(* Logix 5000 project; controller Reto1 vendor 1 type 14 code 156 rev 30.11; software revision 30.00 *)

TASK MainTask (continuous, watchdog 500 ms) : MainProgram

MODULES
   Local : vendor 1 type 14 code 156 (Compact 0, rev 30.11)
END_MODULES

VAR_GLOBAL   (* controller tags *)
   C0 : BOOL;   // OK_INITIALIZATION
   C1 : BOOL;   // OK_STSTEM_ON
   C2 : BOOL;   // OK_POS_TAPA
   C3 : BOOL;   // OK_POS_BASE
   C4 : BOOL;   // OK_FORMADO
   C5 : BOOL;   // OK_FORMADO2
   C6 : BOOL;   // OK_RESET_PROCESS
   CONT_CAJAS : COUNTER := (PRE := 10);
   E0 : BOOL;   // INITIALIZATION
   E1 : BOOL;   // STSTEM_ON
   E2 : BOOL;   // POS_TAPA
   E3 : BOOL;   // POS_BASE
   E4 : BOOL;   // FORMADO
   E5 : BOOL;   // FORMADO2
   E6 : BOOL;   // RESET_PROCESS
   ENT_BASE : BOOL;
   ENT_LID : BOOL;
   ES : BOOL;   // Help Emergency Stop
   GD_IN_0 : BOOL;   // GD_MOVING_X
   GD_IN_1 : BOOL;   // GD_MOVING_Z
   GD_IN_10 : BOOL;   // START_ALL
   GD_IN_11 : BOOL;   // RESET
   GD_IN_12 : BOOL;   // STOP_ALL
   GD_IN_13 : BOOL;   // GD Emergency Stop
   GD_IN_2 : BOOL;   // ITEM_DETECTER
   GD_IN_3 : BOOL;   // LID_AT_PLACE
   GD_IN_4 : BOOL;   // GD_LID_CLAMPED
   GD_IN_5 : BOOL;   // POS_LIMIT_LIDS
   GD_IN_6 : BOOL;   // BASE_AT_PLACE
   GD_IN_7 : BOOL;   // GD_BASE_CLAMPED
   GD_IN_8 : BOOL;   // POS_LIMIT_BASES
   GD_IN_9 : BOOL;   // GD_PART_LEAVING
   GD_OUT_0 : BOOL;   // MOVE_X
   GD_OUT_1 : BOOL;   // MOVE_Z
   GD_OUT_10 : BOOL;   // RESET_LIGHT
   GD_OUT_11 : BOOL;   // STOP_LIGHT
   GD_OUT_2 : BOOL;   // GRAB
   GD_OUT_3 : BOOL;   // LIDS_CONVEYOR
   GD_OUT_4 : BOOL;   // CLAMP_LID
   GD_OUT_5 : BOOL;   // GD_LID_POS_RAISED
   GD_OUT_6 : BOOL;   // BASES_CONVEYOR
   GD_OUT_7 : BOOL;   // CLAMP_BASE
   GD_OUT_8 : BOOL;   // GD_BASE_POS_RAISED
   GD_OUT_9 : BOOL;   // START_LIGHT
   INT1 : BOOL;   // INT1
   ONS_GRAB_OFF : BOOL;
   ONS_INIT_E4 : BOOL;
   ONS_ITEM_DETECTED : BOOL;
   ONS_MX : BOOL;
   ONS_MZ2 : BOOL;
   ONS_OK_FORMADO : BOOL;
   OSF_BASE_IN : BOOL;
   OSF_BASE_OUT : BOOL;
   OSF_BASE_RAISED_ON : BOOL;
   OSF_BASE_RAISED_OUT : BOOL;
   OSF_GRAB_IN : BOOL;
   OSF_GRAB_OUT : BOOL;
   OSF_LID_IN : BOOL;
   OSF_LID_OUT : BOOL;
   OSR_BASE_RAISED_ON : BOOL;
   OSR_BASE_RAISED_OUT : BOOL;
   OSR_FORMADO_IN : BOOL;
   OSR_FORMADO_OUT : BOOL;
   OSR_GRAB_IN : BOOL;
   OSR_GRAB_OFF : BOOL;
   P1 : BOOL;   // TOGGLE BIT
   PC_GOFF : BOOL;
   PC_HZ1 : BOOL;
   PC_HZ2 : BOOL;
   PC_MX : BOOL;
   TB : BOOL;   // TOGGLE_BIT
   TB1 : BOOL;
   TB2 : BOOL;
   TB_E2 : BOOL;
   TB_GRAB : BOOL;
   TB_GRAB_OFF : BOOL;
   TB_HX : BOOL;
   TB_HZ : BOOL;
   TB_HZ_2 : BOOL;
   TB_X : BOOL;
   TB_Z1 : BOOL;
   TB_Z2 : BOOL;
   TIMER_GRAB_OFF : TIMER := (PRE := 250);
   TIMER_HX : TIMER := (PRE := 250);
   TIMER_MZ2 : TIMER := (PRE := 250);
   TIMER_OK_FORMADO : TIMER := (PRE := 250);
   TON_BASE : TIMER := (PRE := 100);
   TON_IE4 : TIMER := (PRE := 500);
   TON_LEAVING : TIMER := (PRE := 500);
   TON_LID : TIMER := (PRE := 100);
END_VAR

PROGRAM MainProgram   (* main routine MainRoutine *)

ROUTINE A_SETUP   (* ladder *)
   0 (stored rung type 13): ;
END_ROUTINE

ROUTINE B_PREPARING   (* ladder *)
   0 (stored rung type 13): ;
END_ROUTINE

ROUTINE C_FORMING   (* ladder *)
END_ROUTINE

ROUTINE MainRoutine   (* ladder *)
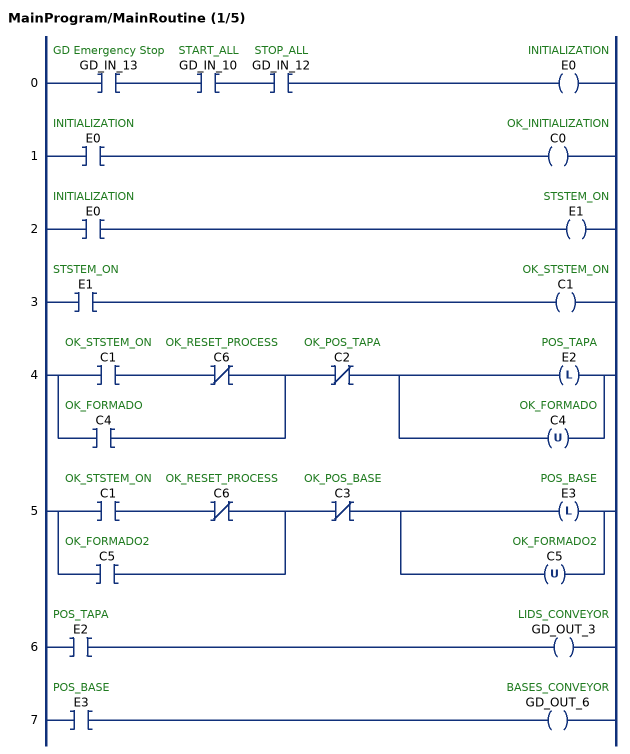
   0: XIC(GD_IN_13)XIC(GD_IN_10)XIC(GD_IN_12)OTE(E0);
   1: XIC(E0)OTE(C0);
   2: XIC(E0)OTE(E1);
   3: XIC(E1)OTE(C1);
   4: [XIC(C1) XIO(C6) ,XIC(C4) ]XIO(C2)[OTL(E2) ,OTU(C4) ];
   5: [XIC(C1) XIO(C6) ,XIC(C5) ]XIO(C3)[OTL(E3) ,OTU(C5) ];
   6: XIC(E2)OTE(GD_OUT_3);
   7: XIC(E3)OTE(GD_OUT_6);
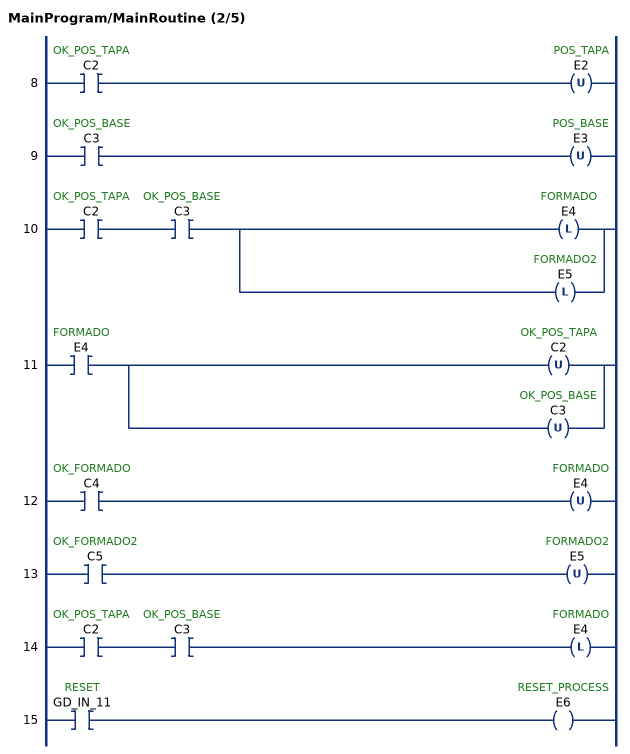
   8: XIC(C2)OTU(E2);
   9: XIC(C3)OTU(E3);
   10: XIC(C2)XIC(C3)[OTL(E4) ,OTL(E5) ];
   11: XIC(E4)[OTU(C2) ,OTU(C3) ];
   12: XIC(C4)OTU(E4);
   13: XIC(C5)OTU(E5);
   14: XIC(C2)XIC(C3)OTL(E4);
   15: XIC(GD_IN_11)OTE(E6);
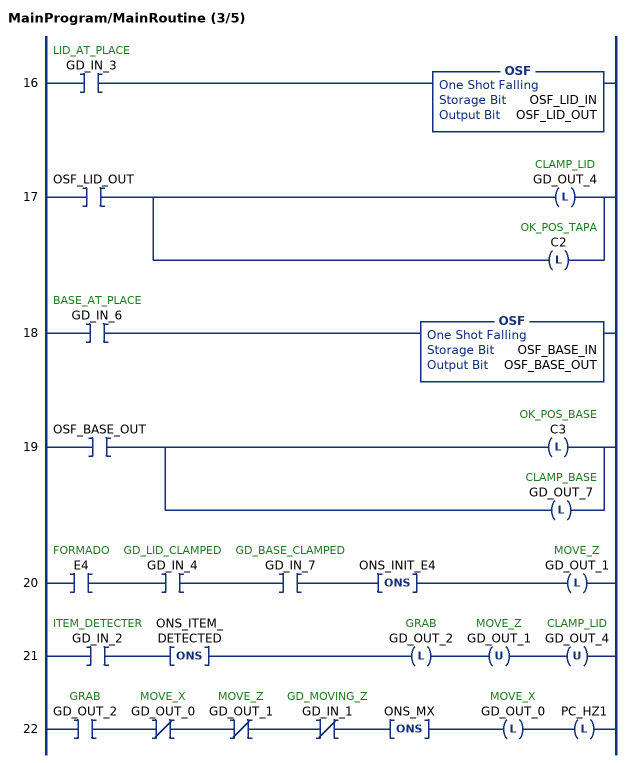
   16: XIC(GD_IN_3)OSF(OSF_LID_IN,OSF_LID_OUT);
   17: XIC(OSF_LID_OUT)[OTL(GD_OUT_4) ,OTL(C2) ];
   18: XIC(GD_IN_6)OSF(OSF_BASE_IN,OSF_BASE_OUT);
   19: XIC(OSF_BASE_OUT)[OTL(C3) ,OTL(GD_OUT_7) ];
   20: XIC(E4)XIC(GD_IN_4)XIC(GD_IN_7)ONS(ONS_INIT_E4)OTL(GD_OUT_1);
   21: XIC(GD_IN_2)ONS(ONS_ITEM_DETECTED)OTL(GD_OUT_2)OTU(GD_OUT_1)OTU(GD_OUT_4);
   22: XIC(GD_OUT_2)XIO(GD_OUT_0)XIO(GD_OUT_1)XIO(GD_IN_1)ONS(ONS_MX)OTL(GD_OUT_0)OTL(PC_HZ1);
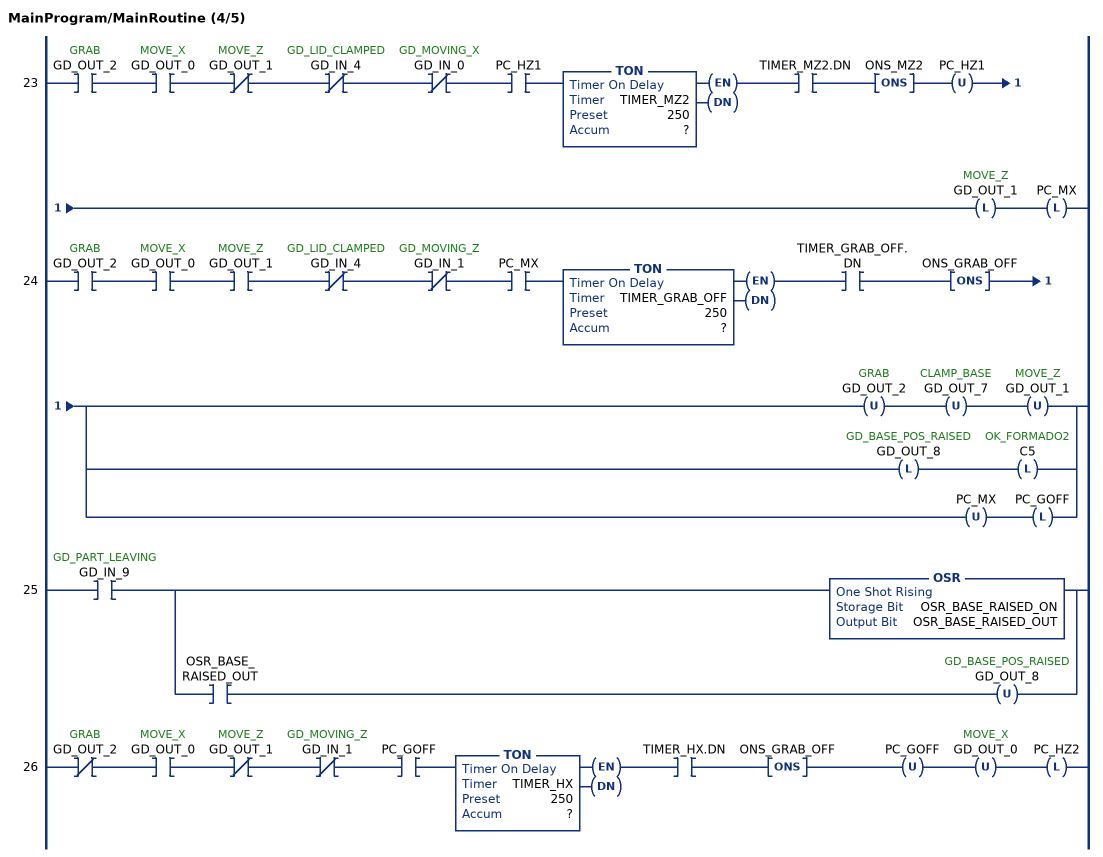
   23: XIC(GD_OUT_2)XIC(GD_OUT_0)XIO(GD_OUT_1)XIO(GD_IN_4)XIO(GD_IN_0)XIC(PC_HZ1)TON(TIMER_MZ2,?,?)XIC(TIMER_MZ2.DN)ONS(ONS_MZ2)OTU(PC_HZ1)OTL(GD_OUT_1)OTL(PC_MX);
   24: XIC(GD_OUT_2)XIC(GD_OUT_0)XIC(GD_OUT_1)XIO(GD_IN_4)XIO(GD_IN_1)XIC(PC_MX)TON(TIMER_GRAB_OFF,?,?)XIC(TIMER_GRAB_OFF.DN)ONS(ONS_GRAB_OFF)[OTU(GD_OUT_2) OTU(GD_OUT_7) OTU(GD_OUT_1) ,[OTL(GD_OUT_8) OTL(C5) ,OTU(PC_MX) OTL(PC_GOFF) ] ];
   25: XIC(GD_IN_9)[OSR(OSR_BASE_RAISED_ON,OSR_BASE_RAISED_OUT) ,XIC(OSR_BASE_RAISED_OUT) OTU(GD_OUT_8) ];
   26: XIO(GD_OUT_2)XIC(GD_OUT_0)XIO(GD_OUT_1)XIO(GD_IN_1)XIC(PC_GOFF)TON(TIMER_HX,?,?)XIC(TIMER_HX.DN)ONS(ONS_GRAB_OFF)OTU(PC_GOFF)OTU(GD_OUT_0)OTL(PC_HZ2);
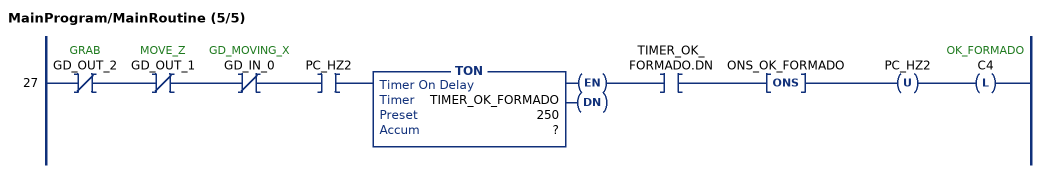
   27: XIO(GD_OUT_2)XIO(GD_OUT_1)XIO(GD_IN_0)XIC(PC_HZ2)TON(TIMER_OK_FORMADO,?,?)XIC(TIMER_OK_FORMADO.DN)ONS(ONS_OK_FORMADO)OTU(PC_HZ2)OTL(C4);
END_ROUTINE

ROUTINE RESET   (* ladder *)
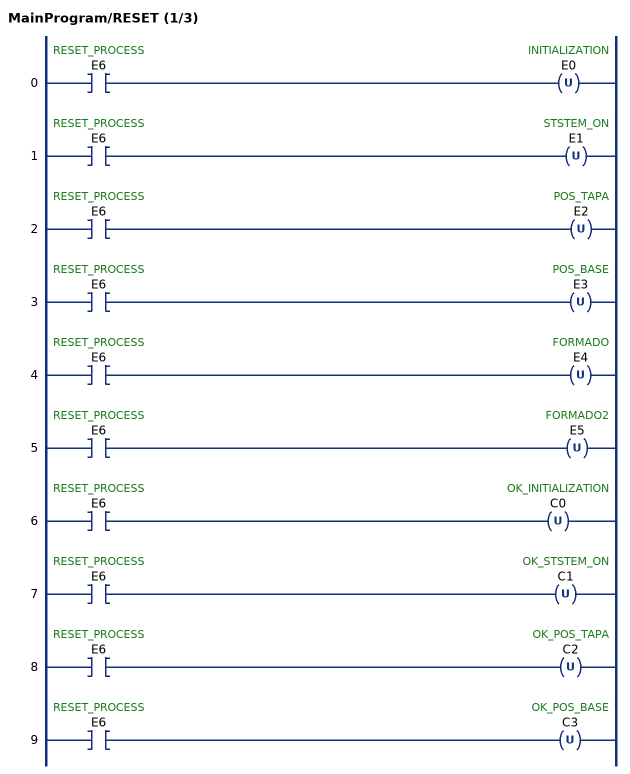
   0: XIC(E6)OTU(E0);
   1: XIC(E6)OTU(E1);
   2: XIC(E6)OTU(E2);
   3: XIC(E6)OTU(E3);
   4: XIC(E6)OTU(E4);
   5: XIC(E6)OTU(E5);
   6: XIC(E6)OTU(C0);
   7: XIC(E6)OTU(C1);
   8: XIC(E6)OTU(C2);
   9: XIC(E6)OTU(C3);
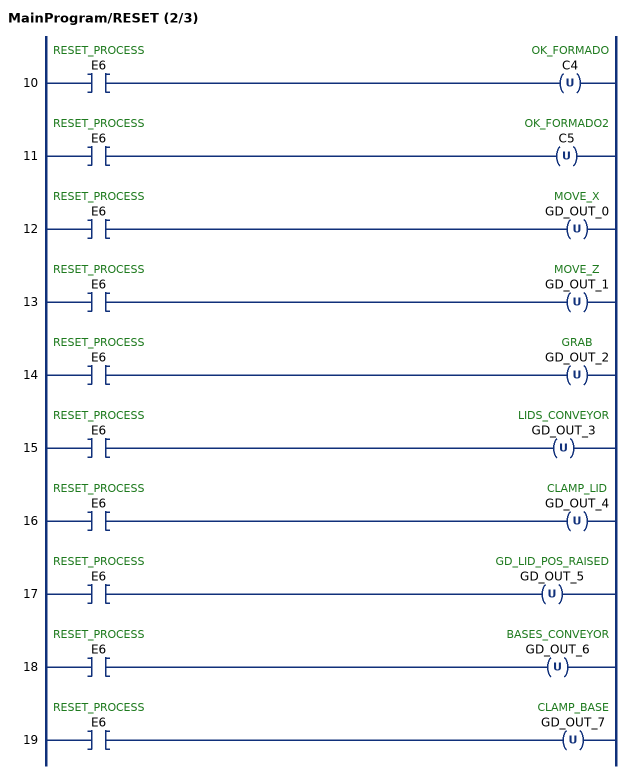
   10: XIC(E6)OTU(C4);
   11: XIC(E6)OTU(C5);
   12: XIC(E6)OTU(GD_OUT_0);
   13: XIC(E6)OTU(GD_OUT_1);
   14: XIC(E6)OTU(GD_OUT_2);
   15: XIC(E6)OTU(GD_OUT_3);
   16: XIC(E6)OTU(GD_OUT_4);
   17: XIC(E6)OTU(GD_OUT_5);
   18: XIC(E6)OTU(GD_OUT_6);
   19: XIC(E6)OTU(GD_OUT_7);
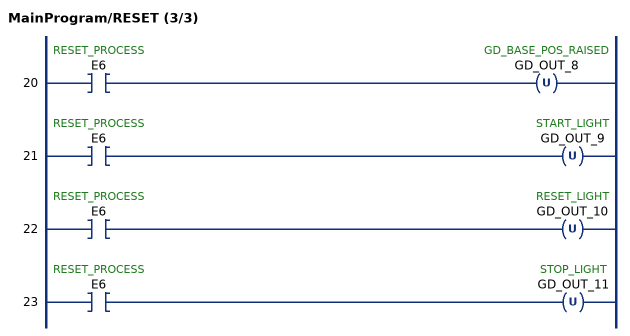
   20: XIC(E6)OTU(GD_OUT_8);
   21: XIC(E6)OTU(GD_OUT_9);
   22: XIC(E6)OTU(GD_OUT_10);
   23: XIC(E6)OTU(GD_OUT_11);
END_ROUTINE
END_PROGRAM
